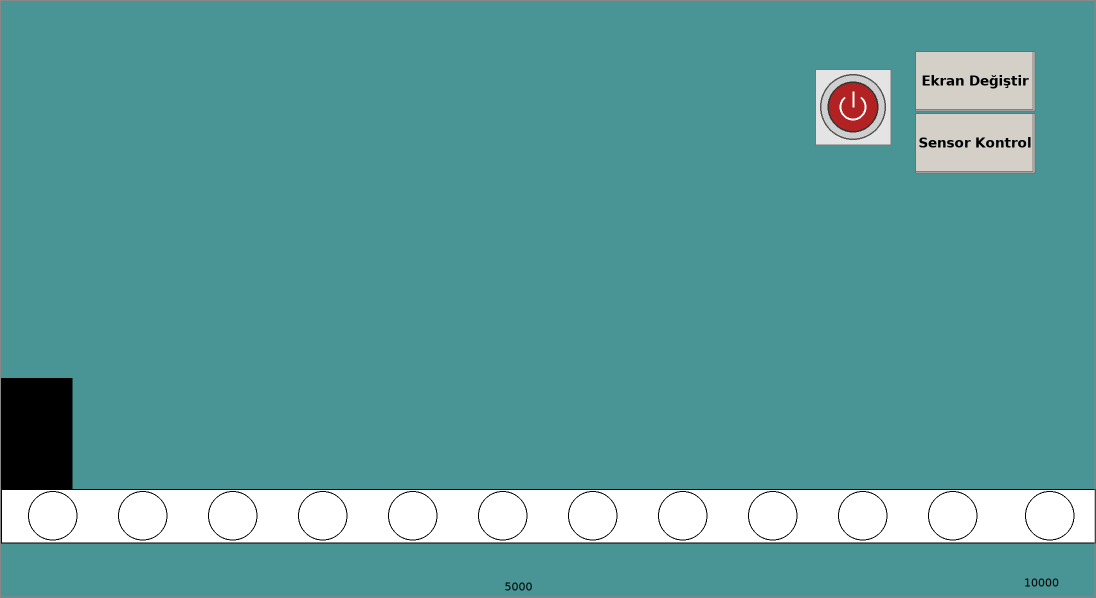
VISUALIZATION VISU_1  // 1096x598
    Rectangle (0,378 72x157)
        p3560616238: MAIN.fPositionVisu
    Group (1,489 1095x54)
        Rectangle (0,0 1095x54)
        Ellipse (27,2 49x49)
        Ellipse (117,2 49x49)
        Ellipse (207,2 49x49)
        Ellipse (297,2 49x49)
        Ellipse (387,2 49x49)
        Ellipse (477,2 49x49)
        Ellipse (567,2 49x49)
        Ellipse (657,2 49x49)
        Ellipse (747,2 49x49)
        Ellipse (837,2 49x49)
        Ellipse (927,2 49x49)
        Ellipse (1024,2 49x49)
    Button (915,51 120x60), "Ekran Değiştir"
        OnMouseClick: change screen: VISU_2
    Button (915,113 120x60), "Sensor Kontrol"
        tap MAIN.bCounter
    PowerSwitch (797,69 112x76), variable: MAIN.bButon, behaviour: TOGGLE, style: Switch-PowerSwitch-Red
    Label (477,576 83x22), "5000"
    Label (1000,572 83x22), "10000"
END_VISUALIZATION

(* stored: Version 1.1.0.1, ProductVersion 3.1.4024.4
   Visu VISU_1: Id {472d9ba1-ff7d-4aac-85fb-3dd1a6c932db} *)
